CELL_RB201_TESTER_SOCKET_D02                        :=          51132       ,
CELL_RB201_TESTER_SOCKET_D03                        :=          51133       ,
CELL_RB201_TESTER_SOCKET_D04                        :=          51134       ,
CELL_RB201_AP                                       :=          51150       ,
CELL_RB201_AP_TH_A01                                :=          51151       ,
CELL_RB201_AP_TH_A02                                :=          51152       ,
CELL_RB201_AP_TH_A03                                :=          51153       ,
CELL_RB201_AP_TH_A04                                :=          51154       ,
CELL_RB201_AP_TH_B01                                :=          51161       ,
CELL_RB201_AP_TH_B02                                :=          51162       ,
CELL_RB201_AP_TH_B03                                :=          51163       ,
CELL_RB201_AP_TH_B04                                :=          51164       ,
CELL_RB201_AP_TH_C01                                :=          51171       ,
CELL_RB201_AP_TH_C02                                :=          51172       ,
CELL_RB201_AP_TH_C03                                :=          51173       ,
CELL_RB201_AP_TH_C04                                :=          51174       ,
CELL_RB201_AP_TH_D01                                :=          51181       ,
CELL_RB201_AP_TH_D02                                :=          51182       ,
CELL_RB201_AP_TH_D03                                :=          51183       ,
CELL_RB201_AP_TH_D04                                :=          51184       ,
CELL_RB301_TESTER                                   :=          51200       ,
CELL_RB301_TESTER_SOCKET_A01                        :=          51201       ,
CELL_RB301_TESTER_SOCKET_A02                        :=          51202       ,
CELL_RB301_TESTER_SOCKET_A03                        :=          51203       ,
CELL_RB301_TESTER_SOCKET_A04                        :=          51204       ,
CELL_RB301_TESTER_SOCKET_B01                        :=          51211       ,
CELL_RB301_TESTER_SOCKET_B02                        :=          51212       ,
CELL_RB301_TESTER_SOCKET_B03                        :=          51213       ,
CELL_RB301_TESTER_SOCKET_B04                        :=          51214       ,
CELL_RB301_TESTER_SOCKET_C01                        :=          51221       ,
CELL_RB301_TESTER_SOCKET_C02                        :=          51222       ,
CELL_RB301_TESTER_SOCKET_C03                        :=          51223       ,
CELL_RB301_TESTER_SOCKET_C04                        :=          51224       ,
CELL_RB301_TESTER_SOCKET_D01                        :=          51231       ,
CELL_RB301_TESTER_SOCKET_D02                        :=          51232       ,
CELL_RB301_TESTER_SOCKET_D03                        :=          51233       ,
CELL_RB301_TESTER_SOCKET_D04                        :=          51234       ,
CELL_RB301_AP                                       :=          51250       ,
CELL_RB301_AP_TH_A01                                :=          51251       ,
CELL_RB301_AP_TH_A02                                :=          51252       ,
CELL_RB301_AP_TH_A03                                :=          51253       ,
CELL_RB301_AP_TH_A04                                :=          51254       ,
CELL_RB301_AP_TH_B01                                :=          51261       ,
CELL_RB301_AP_TH_B02                                :=          51262       ,
CELL_RB301_AP_TH_B03                                :=          51263       ,
CELL_RB301_AP_TH_B04                                :=          51264       ,
CELL_RB301_AP_TH_C01                                :=          51271       ,
CELL_RB301_AP_TH_C02                                :=          51272       ,
CELL_RB301_AP_TH_C03                                :=          51273       ,
CELL_RB301_AP_TH_C04                                :=          51274       ,
CELL_RB301_AP_TH_D01                                :=          51281       ,
CELL_RB301_AP_TH_D02                                :=          51282       ,
CELL_RB301_AP_TH_D03                                :=          51283       ,
CELL_RB301_AP_TH_D04                                :=          51284       ,
CELL_RB401_TESTER                                   :=          51300       ,
CELL_RB401_TESTER_SOCKET_A01                        :=          51301       ,
CELL_RB401_TESTER_SOCKET_A02                        :=          51302       ,
CELL_RB401_TESTER_SOCKET_A03                        :=          51303       ,
CELL_RB401_TESTER_SOCKET_A04                        :=          51304       ,
CELL_RB401_TESTER_SOCKET_B01                        :=          51311       ,
CELL_RB401_TESTER_SOCKET_B02                        :=          51312       ,
CELL_RB401_TESTER_SOCKET_B03                        :=          51313       ,
CELL_RB401_TESTER_SOCKET_B04                        :=          51314       ,
CELL_RB401_TESTER_SOCKET_C01                        :=          51321       ,
CELL_RB401_TESTER_SOCKET_C02                        :=          51322       ,
CELL_RB401_TESTER_SOCKET_C03                        :=          51323       ,
CELL_RB401_TESTER_SOCKET_C04                        :=          51324       ,
CELL_RB401_TESTER_SOCKET_D01                        :=          51331       ,
CELL_RB401_TESTER_SOCKET_D02                        :=          51332       ,
CELL_RB401_TESTER_SOCKET_D03                        :=          51333       ,
CELL_RB401_TESTER_SOCKET_D04                        :=          51334       ,
CELL_RB401_AP                                       :=          51350       ,
CELL_RB401_AP_TH_A01                                :=          51351       ,
CELL_RB401_AP_TH_A02                                :=          51352       ,
CELL_RB401_AP_TH_A03                                :=          51353       ,
CELL_RB401_AP_TH_A04                                :=          51354       ,
CELL_RB401_AP_TH_B01                                :=          51361       ,
CELL_RB401_AP_TH_B02                                :=          51362       ,
CELL_RB401_AP_TH_B03                                :=          51363       ,
CELL_RB401_AP_TH_B04                                :=          51364       ,
CELL_RB401_AP_TH_C01                                :=          51371       ,
CELL_RB401_AP_TH_C02                                :=          51372       ,
CELL_RB401_AP_TH_C03                                :=          51373       ,
CELL_RB401_AP_TH_C04                                :=          51374       ,
CELL_RB401_AP_TH_D01                                :=          51381       ,
CELL_RB401_AP_TH_D02                                :=          51382       ,
CELL_RB401_AP_TH_D03                                :=          51383       ,
CELL_RB401_AP_TH_D04                                :=          51384       ,
CELL_RB501_TESTER                                   :=          51400       ,
CELL_RB501_TESTER_SOCKET_A01                        :=          51401       ,
CELL_RB501_TESTER_SOCKET_A02                        :=          51402       ,
CELL_RB501_TESTER_SOCKET_A03                        :=          51403       ,
CELL_RB501_TESTER_SOCKET_A04                        :=          51404       ,
CELL_RB501_TESTER_SOCKET_B01                        :=          51411       ,
CELL_RB501_TESTER_SOCKET_B02                        :=          51412       ,
CELL_RB501_TESTER_SOCKET_B03                        :=          51413       ,
CELL_RB501_TESTER_SOCKET_B04                        :=          51414       ,
CELL_RB501_TESTER_SOCKET_C01                        :=          51421       ,
CELL_RB501_TESTER_SOCKET_C02                        :=          51422       ,
CELL_RB501_TESTER_SOCKET_C03                        :=          51423       ,
CELL_RB501_TESTER_SOCKET_C04                        :=          51424       ,
CELL_RB501_TESTER_SOCKET_D01                        :=          51431       ,
CELL_RB501_TESTER_SOCKET_D02                        :=          51432       ,
CELL_RB501_TESTER_SOCKET_D03                        :=          51433       ,
CELL_RB501_TESTER_SOCKET_D04                        :=          51434       ,
CELL_RB501_AP                                       :=          51450       ,
CELL_RB501_AP_TH_A01                                :=          51451       ,
CELL_RB501_AP_TH_A02                                :=          51452       ,
CELL_RB501_AP_TH_A03                                :=          51453       ,
CELL_RB501_AP_TH_A04                                :=          51454       ,
CELL_RB501_AP_TH_B01                                :=          51461       ,
CELL_RB501_AP_TH_B02                                :=          51462       ,
CELL_RB501_AP_TH_B03                                :=          51463       ,
CELL_RB501_AP_TH_B04                                :=          51464       ,
CELL_RB501_AP_TH_C01                                :=          51471       ,
CELL_RB501_AP_TH_C02                                :=          51472       ,
CELL_RB501_AP_TH_C03                                :=          51473       ,
CELL_RB501_AP_TH_C04                                :=          51474       ,
CELL_RB501_AP_TH_D01                                :=          51481       ,
CELL_RB501_AP_TH_D02                                :=          51482       ,
CELL_RB501_AP_TH_D03                                :=          51483       ,
CELL_RB501_AP_TH_D04                                :=          51484       ,
CELL_RB601_TESTER                                   :=          51500       ,
CELL_RB601_TESTER_SOCKET_A01                        :=          51501       ,
CELL_RB601_TESTER_SOCKET_A02                        :=          51502       ,
CELL_RB601_TESTER_SOCKET_A03                        :=          51503       ,
CELL_RB601_TESTER_SOCKET_A04                        :=          51504       ,
CELL_RB601_TESTER_SOCKET_B01                        :=          51511       ,
CELL_RB601_TESTER_SOCKET_B02                        :=          51512       ,
CELL_RB601_TESTER_SOCKET_B03                        :=          51513       ,
CELL_RB601_TESTER_SOCKET_B04                        :=          51514       ,
CELL_RB601_TESTER_SOCKET_C01                        :=          51521       ,
CELL_RB601_TESTER_SOCKET_C02                        :=          51522       ,
CELL_RB601_TESTER_SOCKET_C03                        :=          51523       ,
CELL_RB601_TESTER_SOCKET_C04                        :=          51524       ,
CELL_RB601_TESTER_SOCKET_D01                        :=          51531       ,
CELL_RB601_TESTER_SOCKET_D02                        :=          51532       ,
CELL_RB601_TESTER_SOCKET_D03                        :=          51533       ,
CELL_RB601_TESTER_SOCKET_D04                        :=          51534       ,
CELL_RB601_AP                                       :=          51550       ,
CELL_RB601_AP_TH_A01                                :=          51551       ,
CELL_RB601_AP_TH_A02                                :=          51552       ,
CELL_RB601_AP_TH_A03                                :=          51553       ,
CELL_RB601_AP_TH_A04                                :=          51554       ,
CELL_RB601_AP_TH_B01                                :=          51561       ,
CELL_RB601_AP_TH_B02                                :=          51562       ,
CELL_RB601_AP_TH_B03                                :=          51563       ,
CELL_RB601_AP_TH_B04                                :=          51564       ,
CELL_RB601_AP_TH_C01                                :=          51571       ,
CELL_RB601_AP_TH_C02                                :=          51572       ,
CELL_RB601_AP_TH_C03                                :=          51573       ,
CELL_RB601_AP_TH_C04                                :=          51574       ,
CELL_RB601_AP_TH_D01                                :=          51581       ,
CELL_RB601_AP_TH_D02                                :=          51582       ,
CELL_RB601_AP_TH_D03                                :=          51583       ,
CELL_RB601_AP_TH_D04                                :=          51584       ,
CELL_RC101_TESTER                                   :=          52000       ,
CELL_RC101_TESTER_SOCKET_A01                        :=          52001       ,
CELL_RC101_TESTER_SOCKET_A02                        :=          52002       ,
CELL_RC101_TESTER_SOCKET_A03                        :=          52003       ,
CELL_RC101_TESTER_SOCKET_A04                        :=          52004       ,
CELL_RC101_TESTER_SOCKET_B01                        :=          52011       ,
CELL_RC101_TESTER_SOCKET_B02                        :=          52012       ,
CELL_RC101_TESTER_SOCKET_B03                        :=          52013       ,
CELL_RC101_TESTER_SOCKET_B04                        :=          52014       ,
CELL_RC101_TESTER_SOCKET_C01                        :=          52021       ,
CELL_RC101_TESTER_SOCKET_C02                        :=          52022       ,
CELL_RC101_TESTER_SOCKET_C03                        :=          52023       ,
CELL_RC101_TESTER_SOCKET_C04                        :=          52024       ,
CELL_RC101_TESTER_SOCKET_D01                        :=          52031       ,
CELL_RC101_TESTER_SOCKET_D02                        :=          52032       ,
CELL_RC101_TESTER_SOCKET_D03                        :=          52033       ,
CELL_RC101_TESTER_SOCKET_D04                        :=          52034       ,
CELL_RC101_AP                                       :=          52050       ,
CELL_RC101_AP_TH_A01                                :=          52051       ,
CELL_RC101_AP_TH_A02                                :=          52052       ,
CELL_RC101_AP_TH_A03                                :=          52053       ,
CELL_RC101_AP_TH_A04                                :=          52054       ,
CELL_RC101_AP_TH_B01                                :=          52061       ,
CELL_RC101_AP_TH_B02                                :=          52062       ,
CELL_RC101_AP_TH_B03                                :=          52063       ,
CELL_RC101_AP_TH_B04                                :=          52064       ,
CELL_RC101_AP_TH_C01                                :=          52071       ,
CELL_RC101_AP_TH_C02                                :=          52072       ,
CELL_RC101_AP_TH_C03                                :=          52073       ,
CELL_RC101_AP_TH_C04                                :=          52074       ,
CELL_RC101_AP_TH_D01                                :=          52081       ,
CELL_RC101_AP_TH_D02                                :=          52082       ,
CELL_RC101_AP_TH_D03                                :=          52083       ,
CELL_RC101_AP_TH_D04                                :=          52084       ,
CELL_RC201_TESTER                                   :=          52100       ,
CELL_RC201_TESTER_SOCKET_A01                        :=          52101       ,
CELL_RC201_TESTER_SOCKET_A02                        :=          52102       ,
CELL_RC201_TESTER_SOCKET_A03                        :=          52103       ,
CELL_RC201_TESTER_SOCKET_A04                        :=          52104       ,
CELL_RC201_TESTER_SOCKET_B01                        :=          52111       ,
CELL_RC201_TESTER_SOCKET_B02                        :=          52112       ,
CELL_RC201_TESTER_SOCKET_B03                        :=          52113       ,
CELL_RC201_TESTER_SOCKET_B04                        :=          52114       ,
CELL_RC201_TESTER_SOCKET_C01                        :=          52121       ,
CELL_RC201_TESTER_SOCKET_C02                        :=          52122       ,
CELL_RC201_TESTER_SOCKET_C03                        :=          52123       ,
CELL_RC201_TESTER_SOCKET_C04                        :=          52124       ,
CELL_RC201_TESTER_SOCKET_D01                        :=          52131       ,
CELL_RC201_TESTER_SOCKET_D02                        :=          52132       ,
CELL_RC201_TESTER_SOCKET_D03                        :=          52133       ,
CELL_RC201_TESTER_SOCKET_D04                        :=          52134       ,
CELL_RC201_AP                                       :=          52150       ,
CELL_RC201_AP_TH_A01                                :=          52151       ,
CELL_RC201_AP_TH_A02                                :=          52152       ,
CELL_RC201_AP_TH_A03                                :=          52153       ,
CELL_RC201_AP_TH_A04                                :=          52154       ,
CELL_RC201_AP_TH_B01                                :=          52161       ,
CELL_RC201_AP_TH_B02                                :=          52162       ,
CELL_RC201_AP_TH_B03                                :=          52163       ,
CELL_RC201_AP_TH_B04                                :=          52164       ,
CELL_RC201_AP_TH_C01                                :=          52171       ,
CELL_RC201_AP_TH_C02                                :=          52172       ,
CELL_RC201_AP_TH_C03                                :=          52173       ,
CELL_RC201_AP_TH_C04                                :=          52174       ,
CELL_RC201_AP_TH_D01                                :=          52181       ,
CELL_RC201_AP_TH_D02                                :=          52182       ,
CELL_RC201_AP_TH_D03                                :=          52183       ,
CELL_RC201_AP_TH_D04                                :=          52184       ,
CELL_RC301_TESTER                                   :=          52200       ,
CELL_RC301_TESTER_SOCKET_A01                        :=          52201       ,
CELL_RC301_TESTER_SOCKET_A02                        :=          52202       ,
CELL_RC301_TESTER_SOCKET_A03                        :=          52203       ,
CELL_RC301_TESTER_SOCKET_A04                        :=          52204       ,
CELL_RC301_TESTER_SOCKET_B01                        :=          52211       ,
CELL_RC301_TESTER_SOCKET_B02                        :=          52212       ,
CELL_RC301_TESTER_SOCKET_B03                        :=          52213       ,
CELL_RC301_TESTER_SOCKET_B04                        :=          52214       ,
CELL_RC301_TESTER_SOCKET_C01                        :=          52221       ,
CELL_RC301_TESTER_SOCKET_C02                        :=          52222       ,
CELL_RC301_TESTER_SOCKET_C03                        :=          52223       ,
CELL_RC301_TESTER_SOCKET_C04                        :=          52224       ,
CELL_RC301_TESTER_SOCKET_D01                        :=          52231       ,
CELL_RC301_TESTER_SOCKET_D02                        :=          52232       ,
CELL_RC301_TESTER_SOCKET_D03                        :=          52233       ,
CELL_RC301_TESTER_SOCKET_D04                        :=          52234       ,
CELL_RC301_AP                                       :=          52250       ,
CELL_RC301_AP_TH_A01                                :=          52251       ,
CELL_RC301_AP_TH_A02                                :=          52252       ,
CELL_RC301_AP_TH_A03                                :=          52253       ,
CELL_RC301_AP_TH_A04                                :=          52254       ,
CELL_RC301_AP_TH_B01                                :=          52261       ,
CELL_RC301_AP_TH_B02                                :=          52262       ,
CELL_RC301_AP_TH_B03                                :=          52263       ,
CELL_RC301_AP_TH_B04                                :=          52264       ,
CELL_RC301_AP_TH_C01                                :=          52271       ,
CELL_RC301_AP_TH_C02                                :=          52272       ,
CELL_RC301_AP_TH_C03                                :=          52273       ,
CELL_RC301_AP_TH_C04                                :=          52274       ,
CELL_RC301_AP_TH_D01                                :=          52281       ,
CELL_RC301_AP_TH_D02                                :=          52282       ,
CELL_RC301_AP_TH_D03                                :=          52283       ,
CELL_RC301_AP_TH_D04                                :=          52284       ,
CELL_RC401_TESTER                                   :=          52300       ,
CELL_RC401_TESTER_SOCKET_A01                        :=          52301       ,
CELL_RC401_TESTER_SOCKET_A02                        :=          52302       ,
CELL_RC401_TESTER_SOCKET_A03				        :=          52303       ,
CELL_RC401_TESTER_SOCKET_A04                        :=          52304       ,
CELL_RC401_TESTER_SOCKET_B01                        :=          52311       ,
CELL_RC401_TESTER_SOCKET_B02                        :=          52312       ,
CELL_RC401_TESTER_SOCKET_B03                        :=          52313       ,
CELL_RC401_TESTER_SOCKET_B04                        :=          52314       ,
CELL_RC401_TESTER_SOCKET_C01                        :=          52321       ,
CELL_RC401_TESTER_SOCKET_C02                        :=          52322       ,
CELL_RC401_TESTER_SOCKET_C03                        :=          52323       ,
CELL_RC401_TESTER_SOCKET_C04                        :=          52324       ,
CELL_RC401_TESTER_SOCKET_D01                        :=          52331       ,
CELL_RC401_TESTER_SOCKET_D02                        :=          52332       ,
CELL_RC401_TESTER_SOCKET_D03                        :=          52333       ,
CELL_RC401_TESTER_SOCKET_D04                        :=          52334       ,
CELL_RC401_AP                                       :=          52350       ,
CELL_RC401_AP_TH_A01                                :=          52351       ,
CELL_RC401_AP_TH_A02                                :=          52352       ,
CELL_RC401_AP_TH_A03                                :=          52353       ,
CELL_RC401_AP_TH_A04                                :=          52354       ,
CELL_RC401_AP_TH_B01                                :=          52361       ,
CELL_RC401_AP_TH_B02                                :=          52362       ,
CELL_RC401_AP_TH_B03                                :=          52363       ,
CELL_RC401_AP_TH_B04                                :=          52364       ,
CELL_RC401_AP_TH_C01                                :=          52371       ,
CELL_RC401_AP_TH_C02                                :=          52372       ,
CELL_RC401_AP_TH_C03                                :=          52373       ,
CELL_RC401_AP_TH_C04                                :=          52374       ,
CELL_RC401_AP_TH_D01                                :=          52381       ,
CELL_RC401_AP_TH_D02                                :=          52382       ,
CELL_RC401_AP_TH_D03                                :=          52383       ,
CELL_RC401_AP_TH_D04                                :=          52384       ,
CELL_RC501_TESTER                                   :=          52400       ,
CELL_RC501_TESTER_SOCKET_A01                        :=          52401       ,
CELL_RC501_TESTER_SOCKET_A02                        :=          52402       ,
CELL_RC501_TESTER_SOCKET_A03                        :=          52403       ,
CELL_RC501_TESTER_SOCKET_A04                        :=          52404       ,
CELL_RC501_TESTER_SOCKET_B01                        :=          52411       ,
CELL_RC501_TESTER_SOCKET_B02                        :=          52412       ,
CELL_RC501_TESTER_SOCKET_B03                        :=          52413       ,
CELL_RC501_TESTER_SOCKET_B04                        :=          52414       ,
CELL_RC501_TESTER_SOCKET_C01                        :=          52421       ,
CELL_RC501_TESTER_SOCKET_C02                        :=          52422       ,
CELL_RC501_TESTER_SOCKET_C03                        :=          52423       ,
CELL_RC501_TESTER_SOCKET_C04                        :=          52424       ,
CELL_RC501_TESTER_SOCKET_D01                        :=          52431       ,
CELL_RC501_TESTER_SOCKET_D02                        :=          52432       ,
CELL_RC501_TESTER_SOCKET_D03                        :=          52433       ,
CELL_RC501_TESTER_SOCKET_D04                        :=          52434       ,
CELL_RC501_AP                                       :=          52450       ,
CELL_RC501_AP_TH_A01                                :=          52451       ,
CELL_RC501_AP_TH_A02                                :=          52452       ,
CELL_RC501_AP_TH_A03                                :=          52453       ,
CELL_RC501_AP_TH_A04                                :=          52454       ,
CELL_RC501_AP_TH_B01                                :=          52461       ,
CELL_RC501_AP_TH_B02                                :=          52462       ,
CELL_RC501_AP_TH_B03                                :=          52463       ,
CELL_RC501_AP_TH_B04                                :=          52464       ,
CELL_RC501_AP_TH_C01                                :=          52471       ,
CELL_RC501_AP_TH_C02                                :=          52472       ,
CELL_RC501_AP_TH_C03                                :=          52473       ,
CELL_RC501_AP_TH_C04                                :=          52474       ,
CELL_RC501_AP_TH_D01                                :=          52481       ,
CELL_RC501_AP_TH_D02                                :=          52482       ,
CELL_RC501_AP_TH_D03                                :=          52483       ,
CELL_RC501_AP_TH_D04                                :=          52484       ,
CELL_RC601_TESTER                                   :=          52500       ,
CELL_RC601_TESTER_SOCKET_A01                        :=          52501       ,
CELL_RC601_TESTER_SOCKET_A02                        :=          52502       ,
CELL_RC601_TESTER_SOCKET_A03                        :=          52503       ,
CELL_RC601_TESTER_SOCKET_A04                        :=          52504       ,
CELL_RC601_TESTER_SOCKET_B01                        :=          52511       ,
CELL_RC601_TESTER_SOCKET_B02                        :=          52512       ,
CELL_RC601_TESTER_SOCKET_B03                        :=          52513       ,
CELL_RC601_TESTER_SOCKET_B04                        :=          52514       ,
CELL_RC601_TESTER_SOCKET_C01                        :=          52521       ,
CELL_RC601_TESTER_SOCKET_C02                        :=          52522       ,
CELL_RC601_TESTER_SOCKET_C03                        :=          52523       ,
CELL_RC601_TESTER_SOCKET_C04                        :=          52524       ,
CELL_RC601_TESTER_SOCKET_D01                        :=          52531       ,
CELL_RC601_TESTER_SOCKET_D02                        :=          52532       ,
CELL_RC601_TESTER_SOCKET_D03                        :=          52533       ,
CELL_RC601_TESTER_SOCKET_D04                        :=          52534       ,
CELL_RC601_AP                                       :=          52550       ,
CELL_RC601_AP_TH_A01                                :=          52551       ,
CELL_RC601_AP_TH_A02                                :=          52552       ,
CELL_RC601_AP_TH_A03                                :=          52553       ,
CELL_RC601_AP_TH_A04                                :=          52554       ,
CELL_RC601_AP_TH_B01                                :=          52561       ,
CELL_RC601_AP_TH_B02                                :=          52562       ,
CELL_RC601_AP_TH_B03                                :=          52563       ,
CELL_RC601_AP_TH_B04                                :=          52564       ,
CELL_RC601_AP_TH_C01                                :=          52571       ,
CELL_RC601_AP_TH_C02                                :=          52572       ,
CELL_RC601_AP_TH_C03                                :=          52573       ,
CELL_RC601_AP_TH_C04                                :=          52574       ,
CELL_RC601_AP_TH_D01                                :=          52581       ,
CELL_RC601_AP_TH_D02                                :=          52582       ,
CELL_RC601_AP_TH_D03                                :=          52583       ,
CELL_RC601_AP_TH_D04                                :=          52584       ,
CELL_LA101_TIERII                                   :=          54090       ,
CELL_LA201_TIERII                                   :=          54091       ,
CELL_LA301_TIERII                                   :=          54092       ,
CELL_LA401_TIERII                                   :=          54093       ,
CELL_LA501_TIERII                                   :=          54094       ,
CELL_LA601_TIERII                                   :=          54095       ,
CELL_LB101_TIERII                                   :=          54096       ,
CELL_LB201_TIERII                                   :=          54097       ,
CELL_LB301_TIERII                                   :=          54098       ,
CELL_LB401_TIERII                                   :=          54099       ,
CELL_LB501_TIERII                                   :=          54100       ,
CELL_LB601_TIERII                                   :=          54101       ,
CELL_LC101_TIERII                                   :=          54102       ,
CELL_LC201_TIERII                                   :=          54103       ,
CELL_LC301_TIERII                                   :=          54104       ,
CELL_LC401_TIERII                                   :=          54105       ,
CELL_LC501_TIERII                                   :=          54106       ,
CELL_LC601_TIERII                                   :=          54107       ,
CELL_RA101_TIERII                                   :=          54108       ,
CELL_RA201_TIERII                                   :=          54109       ,
CELL_RA301_TIERII                                   :=          54110       ,
CELL_RA401_TIERII                                   :=          54111       ,
CELL_RA501_TIERII                                   :=          54112       ,
CELL_RA601_TIERII                                   :=          54113       ,
CELL_RB101_TIERII                                   :=          54114       ,
CELL_RB201_TIERII                                   :=          54115       ,
CELL_RB301_TIERII                                   :=          54116       ,
CELL_RB401_TIERII                                   :=          54117       ,
CELL_RB501_TIERII                                   :=          54118       ,
CELL_RB601_TIERII                                   :=          54119       ,
CELL_RC101_TIERII                                   :=          54120       ,
CELL_RC201_TIERII                                   :=          54121       ,
CELL_RC301_TIERII                                   :=          54122       ,
CELL_RC401_TIERII                                   :=          54123       ,
CELL_RC501_TIERII                                   :=          54124       ,
CELL_RC601_TIERII                                   :=          54125       

(*
	//New 												  
	NA                                              :=      0    		,
	Standby                                         :=      1           ,
	IOLP                                            :=      2           ,
	PNB                                             :=      3           ,
	TBOT                                            :=      4           ,
	LP_VISIONSHUTTLE_L                              :=      1500        ,
	LP_VISIONSHUTTLE_R                              :=      1600        ,
	LP_LE                                           :=      1900        ,
	LP_L01                                          :=      1901        ,
	LP_L02                                          :=      1902        ,
	LP_RE                                           :=      1903        ,
	LP_R01                                          :=      1904        ,
	LP_R02                                          :=      1905        ,
	LP_L                                            :=      1910        ,
	LP_R                                            :=      1911        ,
	LP_LE_STACKER_01                                :=      2000        ,
	LP_LE_STACKER_01_LIFT                           :=      2001        ,
	LP_LE_STACKER_01_STOPPER_01                     :=      2002        ,
	LP_LE_STACKER_01_STOPPER_02                     :=      2003        ,
	LP_LE_STACKER_02                                :=      2050        ,
	LP_LE_STACKER_02_LIFT                           :=      2051        ,
	LP_LE_STACKER_02_STOPPER_01                     :=      2052        ,
	LP_LE_STACKER_02_STOPPER_02                     :=      2053        ,
	LP_LE_CONVEYOR                                  :=      2200        ,
	LP_LE_CONVEYOR_STACKER_01_PRE                   :=      2250        ,
	LP_LE_CONVEYOR_STACKER_01                       :=      2251        ,
	LP_LE_CONVEYOR_STACKER_01_POST                  :=      2252        ,
	LP_LE_CONVEYOR_STACKER_02                       :=      2300        ,
	LP_L01_STACKER_01                               :=      3000        ,
	LP_L01_STACKER_01_LIFT                          :=      3001        ,
	LP_L01_STACKER_01_STOPPER_01                    :=      3002        ,
	LP_L01_STACKER_01_STOPPER_02                    :=      3003        ,
	LP_L01_STACKER_02                               :=      3050        ,
	LP_L01_STACKER_02_LIFT                          :=      3051        ,
	LP_L01_STACKER_02_STOPPER_01                    :=      3052        ,
	LP_L01_STACKER_02_STOPPER_02                    :=      3053        ,
	LP_L01_STACKER_03                               :=      3100        ,
	LP_L01_STACKER_03_LIFT                          :=      3101        ,
	LP_L01_STACKER_03_STOPPER_01                    :=      3102        ,
	LP_L01_STACKER_03_STOPPER_02                    :=      3103        ,
	LP_L01_CONVEYOR_01                              :=      3110        ,
	LP_L01_CONVEYOR_02                              :=      3120        ,
	LP_L01_CONVEYOR_STACKER_01_PRE                  :=      3125        ,
	LP_L01_CONVEYOR_STACKER_01                      :=      3126        ,
	LP_L01_CONVEYOR_STACKER_01_POST                 :=      3127        ,
	LP_L01_CONVEYOR_STACKER_02                      :=      3128        ,
	LP_L01_CONVEYOR_STACKER_02_POST                 :=      3129        ,
	LP_L01_EPORT                                    :=      3130        ,
	LP_L01_EPORT_STANDBY                            :=      3131        ,
	LP_L01_EPORT_STOPPER_01                         :=      3132        ,
	LP_L01_EPORT_STOPPER_02                         :=      3133        ,
	LP_L01_VISION                                   :=      3140        ,
	LP_L01_UPORT                                    :=      3151        ,
	LP_L02_STACKER_01                               :=      3200        ,
	LP_L02_STACKER_01_LIFT                          :=      3201        ,
	LP_L02_STACKER_01_STOPPER_01                    :=      3202        ,
	LP_L02_STACKER_01_STOPPER_02                    :=      3203        ,
	LP_L02_STACKER_02                               :=      3250        ,
	LP_L02_STACKER_02_LIFT                          :=      3251        ,
	LP_L02_STACKER_02_STOPPER_01                    :=      3252        ,
	LP_L02_STACKER_02_STOPPER_02                    :=      3253        ,
	LP_L02_STACKER_03                               :=      3300        ,
	LP_L02_STACKER_03_LIFT                          :=      3301        ,
	LP_L02_STACKER_03_STOPPER_01                    :=      3302        ,
	LP_L02_STACKER_03_STOPPER_02                    :=      3303        ,
	LP_L02_CONVEYOR_01                              :=      3310        ,
	LP_L02_CONVEYOR_02                              :=      3320        ,
	LP_L02_CONVEYOR_STACKER_01_PRE                  :=      3325        ,
	LP_L02_CONVEYOR_STACKER_01                      :=      3326        ,
	LP_L02_CONVEYOR_STACKER_01_POST                 :=      3327        ,
	LP_L02_CONVEYOR_STACKER_02                      :=      3328        ,
	LP_L02_CONVEYOR_STACKER_02_POST                 :=      3329        ,
	LP_L02_EPORT                                    :=      3330        ,
	LP_L02_EPORT_STANDBY                            :=      3331        ,
	LP_L02_EPORT_STOPPER_01                         :=      3332        ,
	LP_L02_EPORT_STOPPER_02                         :=      3333        ,
	LP_L02_VISION                                   :=      3340        ,
	LP_L02_UPORT                                    :=      3351        ,
	LP_RE_STACKER_01                                :=      4000        ,
	LP_RE_STACKER_01_LIFT                           :=      4001        ,
	LP_RE_STACKER_01_STOPPER_01                     :=      4002        ,
	LP_RE_STACKER_01_STOPPER_02                     :=      4003        ,
	LP_RE_STACKER_02                                :=      4050        ,
	LP_RE_STACKER_02_LIFT                           :=      4051        ,
	LP_RE_STACKER_02_STOPPER_01                     :=      4052        ,
	LP_RE_STACKER_02_STOPPER_02                     :=      4053        ,
	LP_RE_CONVEYOR                                  :=      4200        ,
	LP_RE_CONVEYOR_STACKER_01_PRE                   :=      4250        ,
	LP_RE_CONVEYOR_STACKER_01                       :=      4251        ,
	LP_RE_CONVEYOR_STACKER_01_POST                  :=      4252        ,
	LP_RE_CONVEYOR_STACKER_02                       :=      4300        ,
	LP_R01_STACKER_01                               :=      5000        ,
	LP_R01_STACKER_01_LIFT                          :=      5001        ,
	LP_R01_STACKER_01_STOPPER_01                    :=      5002        ,
	LP_R01_STACKER_01_STOPPER_02                    :=      5003        ,
	LP_R01_STACKER_02                               :=      5050        ,
	LP_R01_STACKER_02_LIFT                          :=      5051        ,
	LP_R01_STACKER_02_STOPPER_01                    :=      5052        ,
	LP_R01_STACKER_02_STOPPER_02                    :=      5053        ,
	LP_R01_STACKER_03                               :=      5100        ,
	LP_R01_STACKER_03_LIFT                          :=      5101        ,
	LP_R01_STACKER_03_STOPPER_01                    :=      5102        ,
	LP_R01_STACKER_03_STOPPER_02                    :=      5103        ,
	LP_R01_CONVEYOR_01                              :=      5110        ,
	LP_R01_CONVEYOR_02                              :=      5120        ,
	LP_R01_CONVEYOR_STACKER_01_PRE                  :=      5125        ,
	LP_R01_CONVEYOR_STACKER_01                      :=      5126        ,
	LP_R01_CONVEYOR_STACKER_01_POST                 :=      5127        ,
	LP_R01_CONVEYOR_STACKER_02                      :=      5128        ,
	LP_R01_CONVEYOR_STACKER_02_POST                 :=      5129        ,
	LP_R01_EPORT                                    :=      5130        ,
	LP_R01_EPORT_STANDBY                            :=      5131        ,
	LP_R01_EPORT_STOPPER_01                         :=      5132        ,
	LP_R01_EPORT_STOPPER_02                         :=      5133        ,
	LP_R01_VISION                                   :=      5140        ,
	LP_R01_UPORT                                    :=      5151        ,
	LP_R02_STACKER_01                               :=      5200        ,
	LP_R02_STACKER_01_LIFT                          :=      5201        ,
	LP_R02_STACKER_01_STOPPER_01                    :=      5202        ,
	LP_R02_STACKER_01_STOPPER_02                    :=      5203        ,
	LP_R02_STACKER_02                               :=      5250        ,
	LP_R02_STACKER_02_LIFT                          :=      5251        ,
	LP_R02_STACKER_02_STOPPER_01                    :=      5252        ,
	LP_R02_STACKER_02_STOPPER_02                    :=      5253        ,
	LP_R02_STACKER_03                               :=      5300        ,
	LP_R02_STACKER_03_LIFT                          :=      5301        ,
	LP_R02_STACKER_03_STOPPER_01                    :=      5302        ,
	LP_R02_STACKER_03_STOPPER_02                    :=      5303        ,
	LP_R02_CONVEYOR_01                              :=      5310        ,
	LP_R02_CONVEYOR_02                              :=      5320        ,
	LP_R02_CONVEYOR_STACKER_01_PRE                  :=      5325        ,
	LP_R02_CONVEYOR_STACKER_01                      :=      5326        ,
	LP_R02_CONVEYOR_STACKER_01_POST                 :=      5327        ,
	LP_R02_CONVEYOR_STACKER_02                      :=      5328        ,
	LP_R02_CONVEYOR_STACKER_02_POST                 :=      5329        ,
	LP_R02_EPORT                                    :=      5330        ,
	LP_R02_EPORT_STANDBY                            :=      5331        ,
	LP_R02_EPORT_STOPPER_01                         :=      5332        ,
	LP_R02_EPORT_STOPPER_02                         :=      5333        ,
	LP_R02_VISION                                   :=      5340        ,
	LP_R02_UPORT                                    :=      5351        ,
	TTS                                             :=      10000       ,
	TTS_SHUTTLE_01                                  :=      10100       ,
	TTS_SHUTTLE_01_SERVICE                          :=      10101       ,
	TTS_SHUTTLE_01_PARK                             :=      10102       ,
	TTS_SHUTTLE_01_CONVEYOR                         :=      10103       ,
	TTS_SHUTTLE_02                                  :=      10200       ,
	TTS_SHUTTLE_02_SERVICE                          :=      10201       ,
	TTS_SHUTTLE_02_CONVEYOR                         :=      10202       ,
	TTS_SHUTTLE_03                                  :=      10300       ,
	TTS_SHUTTLE_03_SERVICE                          :=      10301       ,
	TTS_SHUTTLE_03_PARK                             :=      10302       ,
	TTS_SHUTTLE_03_CONVEYOR                         :=      10303       ,
	PNB_DOOR_TOP_LEFT                               :=      20001       ,
	PNB_DOOR_TOP_RIGHT                              :=      20002       ,
	PNB_DOOR_BOTTOM                                 :=      20003       ,
	PNB_LANE_01                                     :=      21000       ,
	PNB_LANE_01_CONVEYOR                            :=      21001       ,
	PNB_LANE_02                                     :=      21050       ,
	PNB_LANE_02_CONVEYOR                            :=      21051       ,
	PNB_LANE_03                                     :=      21150       ,
	PNB_LANE_03_CONVEYOR                            :=      21151       ,
	PNB_LANE_04                                     :=      21200       ,
	PNB_LANE_04_CONVEYOR                            :=      21201       ,
	PNB_LANE_05                                     :=      21350       ,
	PNB_LANE_05_CONVEYOR                            :=      21351       ,
	PNB_LANE_06                                     :=      21400       ,
	PNB_LANE_06_CONVEYOR                            :=      21401       ,
	PNB_LANE_07                                     :=      21450       ,
	PNB_LANE_07_CONVEYOR                            :=      21451       ,
	PNB_LANE_08                                     :=      21500       ,
	PNB_LANE_08_CONVEYOR                            :=      21501       ,
	PNB_GANTRY_01                                   :=      22500       ,
	PNB_GANTRY_01_PARK                              :=      22501       ,
	PNB_UPCAM_L                                     :=      22502       ,
	PNB_RFID_L                                      :=      22503       ,
	PNB_RFID_L_01                                   :=      22504       ,
	PNB_RFID_L_02                                   :=      22505       ,
	PNB_GANTRY_01_SERVICE                           :=      22506       ,
	PNB_GANTRY_01_HEAD_A01                          :=      22550       ,
	PNB_GANTRY_01_HEAD_A02                          :=      22560       ,
	PNB_GANTRY_01_HEAD_A03                          :=      22570       ,
	PNB_GANTRY_01_HEAD_A04                          :=      22580       ,
	PNB_GANTRY_02                                   :=      23000       ,
	PNB_GANTRY_02_PARK                              :=      23001       ,
	PNB_UPCAM_R                                     :=      23002       ,
	PNB_RFID_R                                      :=      23003       ,
	PNB_RFID_R_01                                   :=      23004       ,
	PNB_RFID_R_02                                   :=      23005       ,
	PNB_GANTRY_02_SERVICE                           :=      22506       ,
	PNB_GANTRY_02_HEAD_A01                          :=      23050       ,
	PNB_GANTRY_02_HEAD_A02                          :=      23060       ,
	PNB_GANTRY_02_HEAD_A03                          :=      23070       ,
	PNB_GANTRY_02_HEAD_A04                          :=      23080       ,
	PRECISOR_UL                                     :=      24000       ,
	PRECISOR_UL_CLEAN                               :=      24001       ,
	PRECISOR_UL_01                                  :=      24002       ,
	PRECISOR_UL_02                                  :=      24003       ,
	PRECISOR_UL_CLEAN_READID                        :=      24004       ,
	PRECISOR_UL_01_READID                           :=      24005       ,
	PRECISOR_UL_02_READID                           :=      24006       ,
	PRECISOR_UL_A01_01                              :=      24011       ,
	PRECISOR_UL_A01_02                              :=      24012       ,
	PRECISOR_UL_A02_01                              :=      24021       ,
	PRECISOR_UL_A02_02                              :=      24022       ,
	PRECISOR_UL_A03_01                              :=      24031       ,
	PRECISOR_UL_A03_02                              :=      24032       ,
	PRECISOR_UL_A04_01                              :=      24041       ,
	PRECISOR_UL_A04_02                              :=      24042       ,
	PRECISOR_UL_B01_01                              :=      24061       ,
	PRECISOR_UL_B01_02                              :=      24062       ,
	PRECISOR_UL_B02_01                              :=      24071       ,
	PRECISOR_UL_B02_02                              :=      24072       ,
	PRECISOR_UL_B03_01                              :=      24081       ,
	PRECISOR_UL_B03_02                              :=      24082       ,
	PRECISOR_UL_B04_01                              :=      24091       ,
	PRECISOR_UL_B04_02                              :=      24092       ,
	PRECISOR_UL_C01_01                              :=      24111       ,
	PRECISOR_UL_C01_02                              :=      24112       ,
	PRECISOR_UL_C02_01                              :=      24121       ,
	PRECISOR_UL_C02_02                              :=      24122       ,
	PRECISOR_UL_C03_01                              :=      24131       ,
	PRECISOR_UL_C03_02                              :=      24132       ,
	PRECISOR_UL_C04_01                              :=      24141       ,
	PRECISOR_UL_C04_02                              :=      24142       ,
	PRECISOR_UL_D01_01                              :=      24161       ,
	PRECISOR_UL_D01_02                              :=      24162       ,
	PRECISOR_UL_D02_01                              :=      24171       ,
	PRECISOR_UL_D02_02                              :=      24172       ,
	PRECISOR_UL_D03_01                              :=      24181       ,
	PRECISOR_UL_D03_02                              :=      24182       ,
	PRECISOR_UL_D04_01                              :=      24191       ,
	PRECISOR_UL_D04_02                              :=      24192       ,
	PRECISOR_UR                                     :=      24500       ,
	PRECISOR_UR_CLEAN                               :=      24501       ,
	PRECISOR_UR_01                                  :=      24502       ,
	PRECISOR_UR_02                                  :=      24503       ,
	PRECISOR_UR_CLEAN_READID                        :=      24504       ,
	PRECISOR_UR_01_READID                           :=      24505       ,
	PRECISOR_UR_02_READID                           :=      24506       ,
	PRECISOR_UR_A01_01                              :=      24511       ,
	PRECISOR_UR_A01_02                              :=      24512       ,
	PRECISOR_UR_A02_01                              :=      24521       ,
	PRECISOR_UR_A02_02                              :=      24522       ,
	PRECISOR_UR_A03_01                              :=      24531       ,
	PRECISOR_UR_A03_02                              :=      24532       ,
	PRECISOR_UR_A04_01                              :=      24541       ,
	PRECISOR_UR_A04_02                              :=      24542       ,
	PRECISOR_UR_B01_01                              :=      24561       ,
	PRECISOR_UR_B01_02                              :=      24562       ,
	PRECISOR_UR_B02_01                              :=      24571       ,
	PRECISOR_UR_B02_02                              :=      24572       ,
	PRECISOR_UR_B03_01                              :=      24581       ,
	PRECISOR_UR_B03_02                              :=      24582       ,
	PRECISOR_UR_B04_01                              :=      24591       ,
	PRECISOR_UR_B04_02                              :=      24592       ,
	PRECISOR_UR_C01_01                              :=      24611       ,
	PRECISOR_UR_C01_02                              :=      24612       ,
	PRECISOR_UR_C02_01                              :=      24621       ,
	PRECISOR_UR_C02_02                              :=      24622       ,
	PRECISOR_UR_C03_01                              :=      24631       ,
	PRECISOR_UR_C03_02                              :=      24632       ,
	PRECISOR_UR_C04_01                              :=      24641       ,
	PRECISOR_UR_C04_02                              :=      24642       ,
	PRECISOR_UR_D01_01                              :=      24661       ,
	PRECISOR_UR_D01_02                              :=      24662       ,
	PRECISOR_UR_D02_01                              :=      24671       ,
	PRECISOR_UR_D02_02                              :=      24672       ,
	PRECISOR_UR_D03_01                              :=      24681       ,
	PRECISOR_UR_D03_02                              :=      24682       ,
	PRECISOR_UR_D04_01                              :=      24691       ,
	PRECISOR_UR_D04_02                              :=      24692       ,
	PRECISOR_DL                                     :=      25000       ,
	PRECISOR_DL_CLEAN                               :=      25001       ,
	PRECISOR_DL_01                                  :=      25002       ,
	PRECISOR_DL_02                                  :=      25003       ,
	PRECISOR_DL_CLEAN_READID                        :=      25004       ,
	PRECISOR_DL_01_READID                           :=      25005       ,
	PRECISOR_DL_02_READID                           :=      25006       ,
	PRECISOR_DL_A01_01                              :=      25011       ,
	PRECISOR_DL_A01_02                              :=      25012       ,
	PRECISOR_DL_A02_01                              :=      25021       ,
	PRECISOR_DL_A02_02                              :=      25022       ,
	PRECISOR_DL_A03_01                              :=      25031       ,
	PRECISOR_DL_A03_02                              :=      25032       ,
	PRECISOR_DL_A04_01                              :=      25041       ,
	PRECISOR_DL_A04_02                              :=      25042       ,
	PRECISOR_DL_B01_01                              :=      25061       ,
	PRECISOR_DL_B01_02                              :=      25062       ,
	PRECISOR_DL_B02_01                              :=      25071       ,
	PRECISOR_DL_B02_02                              :=      25072       ,
	PRECISOR_DL_B03_01                              :=      25081       ,
	PRECISOR_DL_B03_02                              :=      25082       ,
	PRECISOR_DL_B04_01                              :=      25091       ,
	PRECISOR_DL_B04_02                              :=      25092       ,
	PRECISOR_DL_C01_01                              :=      25111       ,
	PRECISOR_DL_C01_02                              :=      25112       ,
	PRECISOR_DL_C02_01                              :=      25121       ,
	PRECISOR_DL_C02_02                              :=      25122       ,
	PRECISOR_DL_C03_01                              :=      25131       ,
	PRECISOR_DL_C03_02                              :=      25132       ,
	PRECISOR_DL_C04_01                              :=      25141       ,
	PRECISOR_DL_C04_02                              :=      25142       ,
	PRECISOR_DL_D01_01                              :=      25161       ,
	PRECISOR_DL_D01_02                              :=      25162       ,
	PRECISOR_DL_D02_01                              :=      25171       ,
	PRECISOR_DL_D02_02                              :=      25172       ,
	PRECISOR_DL_D03_01                              :=      25181       ,
	PRECISOR_DL_D03_02                              :=      25182       ,
	PRECISOR_DL_D04_01                              :=      25191       ,
	PRECISOR_DL_D04_02                              :=      25192       ,
	PRECISOR_DR                                     :=      25500       ,
	PRECISOR_DR_CLEAN                               :=      25501       ,
	PRECISOR_DR_01                                  :=      25502       ,
	PRECISOR_DR_02                                  :=      25503       ,
	PRECISOR_DR_CLEAN_READID                        :=      25504       ,
	PRECISOR_DR_01_READID                           :=      25505       ,
	PRECISOR_DR_02_READID                           :=      25506       ,
	PRECISOR_DR_A01_01                              :=      25511       ,
	PRECISOR_DR_A01_02                              :=      25512       ,
	PRECISOR_DR_A02_01                              :=      25521       ,
	PRECISOR_DR_A02_02                              :=      25522       ,
	PRECISOR_DR_A03_01                              :=      25531       ,
	PRECISOR_DR_A03_02                              :=      25532       ,
	PRECISOR_DR_A04_01                              :=      25541       ,
	PRECISOR_DR_A04_02                              :=      25542       ,
	PRECISOR_DR_B01_01                              :=      25561       ,
	PRECISOR_DR_B01_02                              :=      25562       ,
	PRECISOR_DR_B02_01                              :=      25571       ,
	PRECISOR_DR_B02_02                              :=      25572       ,
	PRECISOR_DR_B03_01                              :=      25581       ,
	PRECISOR_DR_B03_02                              :=      25582       ,
	PRECISOR_DR_B04_01                              :=      25591       ,
	PRECISOR_DR_B04_02                              :=      25592       ,
	PRECISOR_DR_C01_01                              :=      25611       ,
	PRECISOR_DR_C01_02                              :=      25612       ,
	PRECISOR_DR_C02_01                              :=      25621       ,
	PRECISOR_DR_C02_02                              :=      25622       ,
	PRECISOR_DR_C03_01                              :=      25631       ,
	PRECISOR_DR_C03_02                              :=      25632       ,
	PRECISOR_DR_C04_01                              :=      25641       ,
	PRECISOR_DR_C04_02                              :=      25642       ,
	PRECISOR_DR_D01_01                              :=      25661       ,
	PRECISOR_DR_D01_02                              :=      25662       ,
	PRECISOR_DR_D02_01                              :=      25671       ,
	PRECISOR_DR_D02_02                              :=      25672       ,
	PRECISOR_DR_D03_01                              :=      25681       ,
	PRECISOR_DR_D03_02                              :=      25682       ,
	PRECISOR_DR_D04_01                              :=      25691       ,
	PRECISOR_DR_D04_02                              :=      25692       ,
	TBOT_L                                          :=      30000       ,
	TBOT_L_RFID                                     :=      30001       ,
	TBOT_L_SERVICE                                  :=      30002       ,
	TBOT_L_PARK                                     :=      30003       ,
	TBOT_L_HEAD_A01                                 :=      30020       ,
	TBOT_L_HEAD_A02                                 :=      30040       ,
	TBOT_L_HEAD_A03                                 :=      30060       ,
	TBOT_L_HEAD_A04                                 :=      30080       ,
	TBOT_L_HEAD_B01                                 :=      30100       ,
	TBOT_L_HEAD_B02                                 :=      30120       ,
	TBOT_L_HEAD_B03                                 :=      30140       ,
	TBOT_L_HEAD_B04                                 :=      30160       ,
	TBOT_L_HEAD_C01                                 :=      30180       ,
	TBOT_L_HEAD_C02                                 :=      30200       ,
	TBOT_L_HEAD_C03                                 :=      30220       ,
	TBOT_L_HEAD_C04                                 :=      30240       ,
	TBOT_L_HEAD_D01                                 :=      30260       ,
	TBOT_L_HEAD_D02                                 :=      30280       ,
	TBOT_L_HEAD_D03                                 :=      30300       ,
	TBOT_L_HEAD_D04                                 :=      30320       ,
	TBOT_R                                          :=      30500       ,
	TBOT_R_RFID                                     :=      30501       ,
	TBOT_R_SERVICE                                  :=      30502       ,
	TBOT_R_PARK                                     :=      30503       ,
	TBOT_R_HEAD_A01                                 :=      30520       ,
	TBOT_R_HEAD_A02                                 :=      30540       ,
	TBOT_R_HEAD_A03                                 :=      30560       ,
	TBOT_R_HEAD_A04                                 :=      30580       ,
	TBOT_R_HEAD_B01                                 :=      30600       ,
	TBOT_R_HEAD_B02                                 :=      30620       ,
	TBOT_R_HEAD_B03                                 :=      30640       ,
	TBOT_R_HEAD_B04                                 :=      30660       ,
	TBOT_R_HEAD_C01                                 :=      30680       ,
	TBOT_R_HEAD_C02                                 :=      30700       ,
	TBOT_R_HEAD_C03                                 :=      30720       ,
	TBOT_R_HEAD_C04                                 :=      30740       ,
	TBOT_R_HEAD_D01                                 :=      30760       ,
	TBOT_R_HEAD_D02                                 :=      30780       ,
	TBOT_R_HEAD_D03                                 :=      30800       ,
	TBOT_R_HEAD_D04                                 :=      30820       ,
	COLUMN_LA                                       :=      35000       ,
	COLUMN_LB                                       :=      35100       ,
	COLUMN_LC                                       :=      35200       ,
	COLUMN_RA                                       :=      35300       ,
	COLUMN_RB                                       :=      35400       ,
	COLUMN_RC                                       :=      35500       ,
	LEVEL_LA01                                      :=      36000       ,
	LEVEL_LA02                                      :=      36010       ,
	LEVEL_LA03                                      :=      36020       ,
	LEVEL_LA04                                      :=      36030       ,
	LEVEL_LA05                                      :=      36040       ,
	LEVEL_LA06                                      :=      36050       ,
	LEVEL_LB01                                      :=      36060       ,
	LEVEL_LB02                                      :=      36070       ,
	LEVEL_LB03                                      :=      36080       ,
	LEVEL_LB04                                      :=      36090       ,
	LEVEL_LB05                                      :=      36100       ,
	LEVEL_LB06                                      :=      36110       ,
	LEVEL_LC01                                      :=      36120       ,
	LEVEL_LC02                                      :=      36130       ,
	LEVEL_LC03                                      :=      36140       ,
	LEVEL_LC04                                      :=      36150       ,
	LEVEL_LC05                                      :=      36160       ,
	LEVEL_LC06                                      :=      36170       ,
	LEVEL_RA01                                      :=      37000       ,
	LEVEL_RA02                                      :=      37010       ,
	LEVEL_RA03                                      :=      37020       ,
	LEVEL_RA04                                      :=      37030       ,
	LEVEL_RA05                                      :=      37040       ,
	LEVEL_RA06                                      :=      37050       ,
	LEVEL_RB01                                      :=      37060       ,
	LEVEL_RB02                                      :=      37070       ,
	LEVEL_RB03                                      :=      37080       ,
	LEVEL_RB04                                      :=      37090       ,
	LEVEL_RB05                                      :=      37100       ,
	LEVEL_RB06                                      :=      37110       ,
	LEVEL_RC01                                      :=      37120       ,
	LEVEL_RC02                                      :=      37130       ,
	LEVEL_RC03                                      :=      37140       ,
	LEVEL_RC04                                      :=      37150       ,
	LEVEL_RC05                                      :=      37160       ,
	LEVEL_RC06                                      :=      37170       ,
	CELL_LA101_TESTER                               :=      45000       ,
	CELL_LA101_TESTER_SOCKET_A01                    :=      45001       ,
	CELL_LA101_TESTER_SOCKET_A02                    :=      45002       ,
	CELL_LA101_TESTER_SOCKET_A03                    :=      45003       ,
	CELL_LA101_TESTER_SOCKET_A04                    :=      45004       ,
	CELL_LA101_TESTER_SOCKET_B01                    :=      45011       ,
	CELL_LA101_TESTER_SOCKET_B02                    :=      45012       ,
	CELL_LA101_TESTER_SOCKET_B03                    :=      45013       ,
	CELL_LA101_TESTER_SOCKET_B04                    :=      45014       ,
	CELL_LA101_TESTER_SOCKET_C01                    :=      45021       ,
	CELL_LA101_TESTER_SOCKET_C02                    :=      45022       ,
	CELL_LA101_TESTER_SOCKET_C03                    :=      45023       ,
	CELL_LA101_TESTER_SOCKET_C04                    :=      45024       ,
	CELL_LA101_TESTER_SOCKET_D01                    :=      45031       ,
	CELL_LA101_TESTER_SOCKET_D02                    :=      45032       ,
	CELL_LA101_TESTER_SOCKET_D03                    :=      45033       ,
	CELL_LA101_TESTER_SOCKET_D04                    :=      45034       ,
	CELL_LA101_AP                                   :=      45050       ,
	CELL_LA101_AP_TH_A01                            :=      45051       ,
	CELL_LA101_AP_TH_A02                            :=      45052       ,
	CELL_LA101_AP_TH_A03                            :=      45053       ,
	CELL_LA101_AP_TH_A04                            :=      45054       ,
	CELL_LA101_AP_TH_B01                            :=      45061       ,
	CELL_LA101_AP_TH_B02                            :=      45062       ,
	CELL_LA101_AP_TH_B03                            :=      45063       ,
	CELL_LA101_AP_TH_B04                            :=      45064       ,
	CELL_LA101_AP_TH_C01                            :=      45071       ,
	CELL_LA101_AP_TH_C02                            :=      45072       ,
	CELL_LA101_AP_TH_C03                            :=      45073       ,
	CELL_LA101_AP_TH_C04                            :=      45074       ,
	CELL_LA101_AP_TH_D01                            :=      45081       ,
	CELL_LA101_AP_TH_D02                            :=      45082       ,
	CELL_LA101_AP_TH_D03                            :=      45083       ,
	CELL_LA101_AP_TH_D04                            :=      45084       ,
	CELL_LA201_TESTER                               :=      45100       ,
	CELL_LA201_TESTER_SOCKET_A01                    :=      45101       ,
	CELL_LA201_TESTER_SOCKET_A02                    :=      45102       ,
	CELL_LA201_TESTER_SOCKET_A03                    :=      45103       ,
	CELL_LA201_TESTER_SOCKET_A04                    :=      45104       ,
	CELL_LA201_TESTER_SOCKET_B01                    :=      45111       ,
	CELL_LA201_TESTER_SOCKET_B02                    :=      45112       ,
	CELL_LA201_TESTER_SOCKET_B03                    :=      45113       ,
	CELL_LA201_TESTER_SOCKET_B04                    :=      45114       ,
	CELL_LA201_TESTER_SOCKET_C01                    :=      45121       ,
	CELL_LA201_TESTER_SOCKET_C02                    :=      45122       ,
	CELL_LA201_TESTER_SOCKET_C03                    :=      45123       ,
	CELL_LA201_TESTER_SOCKET_C04                    :=      45124       ,
	CELL_LA201_TESTER_SOCKET_D01                    :=      45131       ,
	CELL_LA201_TESTER_SOCKET_D02                    :=      45132       ,
	CELL_LA201_TESTER_SOCKET_D03                    :=      45133       ,
	CELL_LA201_TESTER_SOCKET_D04                    :=      45134       ,
	CELL_LA201_AP                                   :=      45150       ,
	CELL_LA201_AP_TH_A01                            :=      45151       ,
	CELL_LA201_AP_TH_A02                            :=      45152       ,
	CELL_LA201_AP_TH_A03                            :=      45153       ,
	CELL_LA201_AP_TH_A04                            :=      45154       ,
	CELL_LA201_AP_TH_B01                            :=      45161       ,
	CELL_LA201_AP_TH_B02                            :=      45162       ,
	CELL_LA201_AP_TH_B03                            :=      45163       ,
	CELL_LA201_AP_TH_B04                            :=      45164       ,
	CELL_LA201_AP_TH_C01                            :=      45171       ,
	CELL_LA201_AP_TH_C02                            :=      45172       ,
	CELL_LA201_AP_TH_C03                            :=      45173       ,
	CELL_LA201_AP_TH_C04                            :=      45174       ,
	CELL_LA201_AP_TH_D01                            :=      45181       ,
	CELL_LA201_AP_TH_D02                            :=      45182       ,
	CELL_LA201_AP_TH_D03                            :=      45183       ,
	CELL_LA201_AP_TH_D04                            :=      45184       ,
	CELL_LA301_TESTER                               :=      45200       ,
	CELL_LA301_TESTER_SOCKET_A01                    :=      45201       ,
	CELL_LA301_TESTER_SOCKET_A02                    :=      45202       ,
	CELL_LA301_TESTER_SOCKET_A03                    :=      45203       ,
	CELL_LA301_TESTER_SOCKET_A04                    :=      45204       ,
	CELL_LA301_TESTER_SOCKET_B01                    :=      45211       ,
	CELL_LA301_TESTER_SOCKET_B02                    :=      45212       ,
	CELL_LA301_TESTER_SOCKET_B03                    :=      45213       ,
	CELL_LA301_TESTER_SOCKET_B04                    :=      45214       ,
	CELL_LA301_TESTER_SOCKET_C01                    :=      45221       ,
	CELL_LA301_TESTER_SOCKET_C02                    :=      45222       ,
	CELL_LA301_TESTER_SOCKET_C03                    :=      45223       ,
	CELL_LA301_TESTER_SOCKET_C04                    :=      45224       ,
	CELL_LA301_TESTER_SOCKET_D01                    :=      45231       ,
	CELL_LA301_TESTER_SOCKET_D02                    :=      45232       ,
	CELL_LA301_TESTER_SOCKET_D03                    :=      45233       ,
	CELL_LA301_TESTER_SOCKET_D04                    :=      45234       ,
	CELL_LA301_AP                                   :=      45250       ,
	CELL_LA301_AP_TH_A01                            :=      45251       ,
	CELL_LA301_AP_TH_A02                            :=      45252       ,
	CELL_LA301_AP_TH_A03                            :=      45253       ,
	CELL_LA301_AP_TH_A04                            :=      45254       ,
	CELL_LA301_AP_TH_B01                            :=      45261       ,
	CELL_LA301_AP_TH_B02                            :=      45262       ,
	CELL_LA301_AP_TH_B03                            :=      45263       ,
	CELL_LA301_AP_TH_B04                            :=      45264       ,
	CELL_LA301_AP_TH_C01                            :=      45271       ,
	CELL_LA301_AP_TH_C02                            :=      45272       ,
	CELL_LA301_AP_TH_C03                            :=      45273       ,
	CELL_LA301_AP_TH_C04                            :=      45274       ,
	CELL_LA301_AP_TH_D01                            :=      45281       ,
	CELL_LA301_AP_TH_D02                            :=      45282       ,
	CELL_LA301_AP_TH_D03                            :=      45283       ,
	CELL_LA301_AP_TH_D04                            :=      45284       ,
	CELL_LA401_TESTER                               :=      45300       ,
	CELL_LA401_TESTER_SOCKET_A01                    :=      45301       ,
	CELL_LA401_TESTER_SOCKET_A02                    :=      45302       ,
	CELL_LA401_TESTER_SOCKET_A03                    :=      45303       ,
	CELL_LA401_TESTER_SOCKET_A04                    :=      45304       ,
	CELL_LA401_TESTER_SOCKET_B01                    :=      45311       ,
	CELL_LA401_TESTER_SOCKET_B02                    :=      45312       ,
	CELL_LA401_TESTER_SOCKET_B03                    :=      45313       ,
	CELL_LA401_TESTER_SOCKET_B04                    :=      45314       ,
	CELL_LA401_TESTER_SOCKET_C01                    :=      45321       ,
	CELL_LA401_TESTER_SOCKET_C02                    :=      45322       ,
	CELL_LA401_TESTER_SOCKET_C03                    :=      45323       ,
	CELL_LA401_TESTER_SOCKET_C04                    :=      45324       ,
	CELL_LA401_TESTER_SOCKET_D01                    :=      45331       ,
	CELL_LA401_TESTER_SOCKET_D02                    :=      45332       ,
	CELL_LA401_TESTER_SOCKET_D03                    :=      45333       ,
	CELL_LA401_TESTER_SOCKET_D04                    :=      45334       ,
	CELL_LA401_AP                                   :=      45350       ,
	CELL_LA401_AP_TH_A01                            :=      45351       ,
	CELL_LA401_AP_TH_A02                            :=      45352       ,
	CELL_LA401_AP_TH_A03                            :=      45353       ,
	CELL_LA401_AP_TH_A04                            :=      45354       ,
	CELL_LA401_AP_TH_B01                            :=      45361       ,
	CELL_LA401_AP_TH_B02                            :=      45362       ,
	CELL_LA401_AP_TH_B03                            :=      45363       ,
	CELL_LA401_AP_TH_B04                            :=      45364       ,
	CELL_LA401_AP_TH_C01                            :=      45371       ,
	CELL_LA401_AP_TH_C02                            :=      45372       ,
	CELL_LA401_AP_TH_C03                            :=      45373       ,
	CELL_LA401_AP_TH_C04                            :=      45374       ,
	CELL_LA401_AP_TH_D01                            :=      45381       ,
	CELL_LA401_AP_TH_D02                            :=      45382       ,
	CELL_LA401_AP_TH_D03                            :=      45383       ,
	CELL_LA401_AP_TH_D04                            :=      45384       ,
	CELL_LA501_TESTER                               :=      45400       ,
	CELL_LA501_TESTER_SOCKET_A01                    :=      45401       ,
	CELL_LA501_TESTER_SOCKET_A02                    :=      45402       ,
	CELL_LA501_TESTER_SOCKET_A03                    :=      45403       ,
	CELL_LA501_TESTER_SOCKET_A04                    :=      45404       ,
	CELL_LA501_TESTER_SOCKET_B01                    :=      45411       ,
	CELL_LA501_TESTER_SOCKET_B02                    :=      45412       ,
	CELL_LA501_TESTER_SOCKET_B03                    :=      45413       ,
	CELL_LA501_TESTER_SOCKET_B04                    :=      45414       ,
	CELL_LA501_TESTER_SOCKET_C01                    :=      45421       ,
	CELL_LA501_TESTER_SOCKET_C02                    :=      45422       ,
	CELL_LA501_TESTER_SOCKET_C03                    :=      45423       ,
	CELL_LA501_TESTER_SOCKET_C04                    :=      45424       ,
	CELL_LA501_TESTER_SOCKET_D01                    :=      45431       ,
	CELL_LA501_TESTER_SOCKET_D02                    :=      45432       ,
	CELL_LA501_TESTER_SOCKET_D03                    :=      45433       ,
	CELL_LA501_TESTER_SOCKET_D04                    :=      45434       ,
	CELL_LA501_AP                                   :=      45450       ,
	CELL_LA501_AP_TH_A01                            :=      45451       ,
	CELL_LA501_AP_TH_A02                            :=      45452       ,
	CELL_LA501_AP_TH_A03                            :=      45453       ,
	CELL_LA501_AP_TH_A04                            :=      45454       ,
	CELL_LA501_AP_TH_B01                            :=      45461       ,
	CELL_LA501_AP_TH_B02                            :=      45462       ,
	CELL_LA501_AP_TH_B03                            :=      45463       ,
	CELL_LA501_AP_TH_B04                            :=      45464       ,
	CELL_LA501_AP_TH_C01                            :=      45471       ,
	CELL_LA501_AP_TH_C02                            :=      45472       ,
	CELL_LA501_AP_TH_C03                            :=      45473       ,
	CELL_LA501_AP_TH_C04                            :=      45474       ,
	CELL_LA501_AP_TH_D01                            :=      45481       ,
	CELL_LA501_AP_TH_D02                            :=      45482       ,
	CELL_LA501_AP_TH_D03                            :=      45483       ,
	CELL_LA501_AP_TH_D04                            :=      45484       ,
	CELL_LA601_TESTER                               :=      45500       ,
	CELL_LA601_TESTER_SOCKET_A01                    :=      45501       ,
	CELL_LA601_TESTER_SOCKET_A02                    :=      45502       ,
	CELL_LA601_TESTER_SOCKET_A03                    :=      45503       ,
	CELL_LA601_TESTER_SOCKET_A04                    :=      45504       ,
	CELL_LA601_TESTER_SOCKET_B01                    :=      45511       ,
	CELL_LA601_TESTER_SOCKET_B02                    :=      45512       ,
	CELL_LA601_TESTER_SOCKET_B03                    :=      45513       ,
	CELL_LA601_TESTER_SOCKET_B04                    :=      45514       ,
	CELL_LA601_TESTER_SOCKET_C01                    :=      45521       ,
	CELL_LA601_TESTER_SOCKET_C02                    :=      45522       ,
	CELL_LA601_TESTER_SOCKET_C03                    :=      45523       ,
	CELL_LA601_TESTER_SOCKET_C04                    :=      45524       ,
	CELL_LA601_TESTER_SOCKET_D01                    :=      45531       ,
	CELL_LA601_TESTER_SOCKET_D02                    :=      45532       ,
	CELL_LA601_TESTER_SOCKET_D03                    :=      45533       ,
	CELL_LA601_TESTER_SOCKET_D04                    :=      45534       ,
	CELL_LA601_AP                                   :=      45550       ,
	CELL_LA601_AP_TH_A01                            :=      45551       ,
	CELL_LA601_AP_TH_A02                            :=      45552       ,
	CELL_LA601_AP_TH_A03                            :=      45553       ,
	CELL_LA601_AP_TH_A04                            :=      45554       ,
	CELL_LA601_AP_TH_B01                            :=      45561       ,
	CELL_LA601_AP_TH_B02                            :=      45562       ,
	CELL_LA601_AP_TH_B03                            :=      45563       ,
	CELL_LA601_AP_TH_B04                            :=      45564       ,
	CELL_LA601_AP_TH_C01                            :=      45571       ,
	CELL_LA601_AP_TH_C02                            :=      45572       ,
	CELL_LA601_AP_TH_C03                            :=      45573       ,
	CELL_LA601_AP_TH_C04                            :=      45574       ,
	CELL_LA601_AP_TH_D01                            :=      45581       ,
	CELL_LA601_AP_TH_D02                            :=      45582       ,
	CELL_LA601_AP_TH_D03                            :=      45583       ,
	CELL_LA601_AP_TH_D04                            :=      45584       ,
	CELL_LB101_TESTER                               :=      46000       ,
	CELL_LB101_TESTER_SOCKET_A01                    :=      46001       ,
	CELL_LB101_TESTER_SOCKET_A02                    :=      46002       ,
	CELL_LB101_TESTER_SOCKET_A03                    :=      46003       ,
	CELL_LB101_TESTER_SOCKET_A04                    :=      46004       ,
	CELL_LB101_TESTER_SOCKET_B01                    :=      46011       ,
	CELL_LB101_TESTER_SOCKET_B02                    :=      46012       ,
	CELL_LB101_TESTER_SOCKET_B03                    :=      46013       ,
	CELL_LB101_TESTER_SOCKET_B04                    :=      46014       ,
	CELL_LB101_TESTER_SOCKET_C01                    :=      46021       ,
	CELL_LB101_TESTER_SOCKET_C02                    :=      46022       ,
	CELL_LB101_TESTER_SOCKET_C03                    :=      46023       ,
	CELL_LB101_TESTER_SOCKET_C04                    :=      46024       ,
	CELL_LB101_TESTER_SOCKET_D01                    :=      46031       ,
	CELL_LB101_TESTER_SOCKET_D02                    :=      46032       ,
	CELL_LB101_TESTER_SOCKET_D03                    :=      46033       ,
	CELL_LB101_TESTER_SOCKET_D04                    :=      46034       ,
	CELL_LB101_AP                                   :=      46050       ,
	CELL_LB101_AP_TH_A01                            :=      46051       ,
	CELL_LB101_AP_TH_A02                            :=      46052       ,
	CELL_LB101_AP_TH_A03                            :=      46053       ,
	CELL_LB101_AP_TH_A04                            :=      46054       ,
	CELL_LB101_AP_TH_B01                            :=      46061       ,
	CELL_LB101_AP_TH_B02                            :=      46062       ,
	CELL_LB101_AP_TH_B03                            :=      46063       ,
	CELL_LB101_AP_TH_B04                            :=      46064       ,
	CELL_LB101_AP_TH_C01                            :=      46071       ,
	CELL_LB101_AP_TH_C02                            :=      46072       ,
	CELL_LB101_AP_TH_C03                            :=      46073       ,
	CELL_LB101_AP_TH_C04                            :=      46074       ,
	CELL_LB101_AP_TH_D01                            :=      46081       ,
	CELL_LB101_AP_TH_D02                            :=      46082       ,
	CELL_LB101_AP_TH_D03                            :=      46083       ,
	CELL_LB101_AP_TH_D04                            :=      46084       ,
	CELL_LB201_TESTER                               :=      46100       ,
	CELL_LB201_TESTER_SOCKET_A01                    :=      46101       ,
	CELL_LB201_TESTER_SOCKET_A02                    :=      46102       ,
	CELL_LB201_TESTER_SOCKET_A03                    :=      46103       ,
	CELL_LB201_TESTER_SOCKET_A04                    :=      46104       ,
	CELL_LB201_TESTER_SOCKET_B01                    :=      46111       ,
	CELL_LB201_TESTER_SOCKET_B02                    :=      46112       ,
	CELL_LB201_TESTER_SOCKET_B03                    :=      46113       ,
	CELL_LB201_TESTER_SOCKET_B04                    :=      46114       ,
	CELL_LB201_TESTER_SOCKET_C01                    :=      46121       ,
	CELL_LB201_TESTER_SOCKET_C02                    :=      46122       ,
	CELL_LB201_TESTER_SOCKET_C03                    :=      46123       ,
	CELL_LB201_TESTER_SOCKET_C04                    :=      46124       ,
	CELL_LB201_TESTER_SOCKET_D01                    :=      46131       ,
	CELL_LB201_TESTER_SOCKET_D02                    :=      46132       ,
	CELL_LB201_TESTER_SOCKET_D03                    :=      46133       ,
	CELL_LB201_TESTER_SOCKET_D04                    :=      46134       ,
	CELL_LB201_AP                                   :=      46150       ,
	CELL_LB201_AP_TH_A01                            :=      46151       ,
	CELL_LB201_AP_TH_A02                            :=      46152       ,
	CELL_LB201_AP_TH_A03                            :=      46153       ,
	CELL_LB201_AP_TH_A04                            :=      46154       ,
	CELL_LB201_AP_TH_B01                            :=      46161       ,
	CELL_LB201_AP_TH_B02                            :=      46162       ,
	CELL_LB201_AP_TH_B03                            :=      46163       ,
	CELL_LB201_AP_TH_B04                            :=      46164       ,
	CELL_LB201_AP_TH_C01                            :=      46171       ,
	CELL_LB201_AP_TH_C02                            :=      46172       ,
	CELL_LB201_AP_TH_C03                            :=      46173       ,
	CELL_LB201_AP_TH_C04                            :=      46174       ,
	CELL_LB201_AP_TH_D01                            :=      46181       ,
	CELL_LB201_AP_TH_D02                            :=      46182       ,
	CELL_LB201_AP_TH_D03                            :=      46183       ,
	CELL_LB201_AP_TH_D04                            :=      46184       ,
	CELL_LB301_TESTER                               :=      46200       ,
	CELL_LB301_TESTER_SOCKET_A01                    :=      46201       ,
	CELL_LB301_TESTER_SOCKET_A02                    :=      46202       ,
	CELL_LB301_TESTER_SOCKET_A03                    :=      46203       ,
	CELL_LB301_TESTER_SOCKET_A04                    :=      46204       ,
	CELL_LB301_TESTER_SOCKET_B01                    :=      46211       ,
	CELL_LB301_TESTER_SOCKET_B02                    :=      46212       ,
	CELL_LB301_TESTER_SOCKET_B03                    :=      46213       ,
	CELL_LB301_TESTER_SOCKET_B04                    :=      46214       ,
	CELL_LB301_TESTER_SOCKET_C01                    :=      46221       ,
	CELL_LB301_TESTER_SOCKET_C02                    :=      46222       ,
	CELL_LB301_TESTER_SOCKET_C03                    :=      46223       ,
	CELL_LB301_TESTER_SOCKET_C04                    :=      46224       ,
	CELL_LB301_TESTER_SOCKET_D01                    :=      46231       ,
	CELL_LB301_TESTER_SOCKET_D02                    :=      46232       ,
	CELL_LB301_TESTER_SOCKET_D03                    :=      46233       ,
	CELL_LB301_TESTER_SOCKET_D04                    :=      46234       ,
	CELL_LB301_AP                                   :=      46250       ,
	CELL_LB301_AP_TH_A01                            :=      46251       ,
	CELL_LB301_AP_TH_A02                            :=      46252       ,
	CELL_LB301_AP_TH_A03                            :=      46253       ,
	CELL_LB301_AP_TH_A04                            :=      46254       ,
	CELL_LB301_AP_TH_B01                            :=      46261       ,
	CELL_LB301_AP_TH_B02                            :=      46262       ,
	CELL_LB301_AP_TH_B03                            :=      46263       ,
	CELL_LB301_AP_TH_B04                            :=      46264       ,
	CELL_LB301_AP_TH_C01                            :=      46271       ,
	CELL_LB301_AP_TH_C02                            :=      46272       ,
	CELL_LB301_AP_TH_C03                            :=      46273       ,
	CELL_LB301_AP_TH_C04                            :=      46274       ,
	CELL_LB301_AP_TH_D01                            :=      46281       ,
	CELL_LB301_AP_TH_D02                            :=      46282       ,
	CELL_LB301_AP_TH_D03                            :=      46283       ,
	CELL_LB301_AP_TH_D04                            :=      46284       ,
	CELL_LB401_TESTER                               :=      46300       ,
	CELL_LB401_TESTER_SOCKET_A01                    :=      46301       ,
	CELL_LB401_TESTER_SOCKET_A02                    :=      46302       ,
	CELL_LB401_TESTER_SOCKET_A03                    :=      46303       ,
	CELL_LB401_TESTER_SOCKET_A04                    :=      46304       ,
	CELL_LB401_TESTER_SOCKET_B01                    :=      46311       ,
	CELL_LB401_TESTER_SOCKET_B02                    :=      46312       ,
	CELL_LB401_TESTER_SOCKET_B03                    :=      46313       ,
	CELL_LB401_TESTER_SOCKET_B04                    :=      46314       ,
	CELL_LB401_TESTER_SOCKET_C01                    :=      46321       ,
	CELL_LB401_TESTER_SOCKET_C02                    :=      46322       ,
	CELL_LB401_TESTER_SOCKET_C03                    :=      46323       ,
	CELL_LB401_TESTER_SOCKET_C04                    :=      46324       ,
	CELL_LB401_TESTER_SOCKET_D01                    :=      46331       ,
	CELL_LB401_TESTER_SOCKET_D02                    :=      46332       ,
	CELL_LB401_TESTER_SOCKET_D03                    :=      46333       ,
	CELL_LB401_TESTER_SOCKET_D04                    :=      46334       ,
	CELL_LB401_AP                                   :=      46350       ,
	CELL_LB401_AP_TH_A01                            :=      46351       ,
	CELL_LB401_AP_TH_A02                            :=      46352       ,
	CELL_LB401_AP_TH_A03                            :=      46353       ,
	CELL_LB401_AP_TH_A04                            :=      46354       ,
	CELL_LB401_AP_TH_B01                            :=      46361       ,
	CELL_LB401_AP_TH_B02                            :=      46362       ,
	CELL_LB401_AP_TH_B03                            :=      46363       ,
	CELL_LB401_AP_TH_B04                            :=      46364       ,
	CELL_LB401_AP_TH_C01                            :=      46371       ,
	CELL_LB401_AP_TH_C02                            :=      46372       ,
	CELL_LB401_AP_TH_C03                            :=      46373       ,
	CELL_LB401_AP_TH_C04                            :=      46374       ,
	CELL_LB401_AP_TH_D01                            :=      46381       ,
	CELL_LB401_AP_TH_D02                            :=      46382       ,
	CELL_LB401_AP_TH_D03                            :=      46383       ,
	CELL_LB401_AP_TH_D04                            :=      46384       ,
	CELL_LB501_TESTER                               :=      46400       ,
	CELL_LB501_TESTER_SOCKET_A01                    :=      46401       ,
	CELL_LB501_TESTER_SOCKET_A02                    :=      46402       ,
	CELL_LB501_TESTER_SOCKET_A03                    :=      46403       ,
	CELL_LB501_TESTER_SOCKET_A04                    :=      46404       ,
	CELL_LB501_TESTER_SOCKET_B01                    :=      46411       ,
	CELL_LB501_TESTER_SOCKET_B02                    :=      46412       ,
	CELL_LB501_TESTER_SOCKET_B03                    :=      46413       ,
	CELL_LB501_TESTER_SOCKET_B04                    :=      46414       ,
	CELL_LB501_TESTER_SOCKET_C01                    :=      46421       ,
	CELL_LB501_TESTER_SOCKET_C02                    :=      46422       ,
	CELL_LB501_TESTER_SOCKET_C03                    :=      46423       ,
	CELL_LB501_TESTER_SOCKET_C04                    :=      46424       ,
	CELL_LB501_TESTER_SOCKET_D01                    :=      46431       ,
	CELL_LB501_TESTER_SOCKET_D02                    :=      46432       ,
	CELL_LB501_TESTER_SOCKET_D03                    :=      46433       ,
	CELL_LB501_TESTER_SOCKET_D04                    :=      46434       ,
	CELL_LB501_AP                                   :=      46450       ,
	CELL_LB501_AP_TH_A01                            :=      46451       ,
	CELL_LB501_AP_TH_A02                            :=      46452       ,
	CELL_LB501_AP_TH_A03                            :=      46453       ,
	CELL_LB501_AP_TH_A04                            :=      46454       ,
	CELL_LB501_AP_TH_B01                            :=      46461       ,
	CELL_LB501_AP_TH_B02                            :=      46462       ,
	CELL_LB501_AP_TH_B03                            :=      46463       ,
	CELL_LB501_AP_TH_B04                            :=      46464       ,
	CELL_LB501_AP_TH_C01                            :=      46471       ,
	CELL_LB501_AP_TH_C02                            :=      46472       ,
	CELL_LB501_AP_TH_C03                            :=      46473       ,
	CELL_LB501_AP_TH_C04                            :=      46474       ,
	CELL_LB501_AP_TH_D01                            :=      46481       ,
	CELL_LB501_AP_TH_D02                            :=      46482       ,
	CELL_LB501_AP_TH_D03                            :=      46483       ,
	CELL_LB501_AP_TH_D04                            :=      46484       ,
	CELL_LB601_TESTER                               :=      46500       ,
	CELL_LB601_TESTER_SOCKET_A01                    :=      46501       ,
	CELL_LB601_TESTER_SOCKET_A02                    :=      46502       ,
	CELL_LB601_TESTER_SOCKET_A03                    :=      46503       ,
	CELL_LB601_TESTER_SOCKET_A04                    :=      46504       ,
	CELL_LB601_TESTER_SOCKET_B01                    :=      46511       ,
	CELL_LB601_TESTER_SOCKET_B02                    :=      46512       ,
	CELL_LB601_TESTER_SOCKET_B03                    :=      46513       ,
	CELL_LB601_TESTER_SOCKET_B04                    :=      46514       ,
	CELL_LB601_TESTER_SOCKET_C01                    :=      46521       ,
	CELL_LB601_TESTER_SOCKET_C02                    :=      46522       ,
	CELL_LB601_TESTER_SOCKET_C03                    :=      46523       ,
	CELL_LB601_TESTER_SOCKET_C04                    :=      46524       ,
	CELL_LB601_TESTER_SOCKET_D01                    :=      46531       ,
	CELL_LB601_TESTER_SOCKET_D02                    :=      46532       ,
	CELL_LB601_TESTER_SOCKET_D03                    :=      46533       ,
	CELL_LB601_TESTER_SOCKET_D04                    :=      46534       ,
	CELL_LB601_AP                                   :=      46550       ,
	CELL_LB601_AP_TH_A01                            :=      46551       ,
	CELL_LB601_AP_TH_A02                            :=      46552       ,
	CELL_LB601_AP_TH_A03                            :=      46553       ,
	CELL_LB601_AP_TH_A04                            :=      46554       ,
	CELL_LB601_AP_TH_B01                            :=      46561       ,
	CELL_LB601_AP_TH_B02                            :=      46562       ,
	CELL_LB601_AP_TH_B03                            :=      46563       ,
	CELL_LB601_AP_TH_B04                            :=      46564       ,
	CELL_LB601_AP_TH_C01                            :=      46571       ,
	CELL_LB601_AP_TH_C02                            :=      46572       ,
	CELL_LB601_AP_TH_C03                            :=      46573       ,
	CELL_LB601_AP_TH_C04                            :=      46574       ,
	CELL_LB601_AP_TH_D01                            :=      46581       ,
	CELL_LB601_AP_TH_D02                            :=      46582       ,
	CELL_LB601_AP_TH_D03                            :=      46583       ,
	CELL_LB601_AP_TH_D04                            :=      46584       ,
	CELL_LC101_TESTER                               :=      47000       ,
	CELL_LC101_TESTER_SOCKET_A01                    :=      47001       ,
	CELL_LC101_TESTER_SOCKET_A02                    :=      47002       ,
	CELL_LC101_TESTER_SOCKET_A03                    :=      47003       ,
	CELL_LC101_TESTER_SOCKET_A04                    :=      47004       ,
	CELL_LC101_TESTER_SOCKET_B01                    :=      47011       ,
	CELL_LC101_TESTER_SOCKET_B02                    :=      47012       ,
	CELL_LC101_TESTER_SOCKET_B03                    :=      47013       ,
	CELL_LC101_TESTER_SOCKET_B04                    :=      47014       ,
	CELL_LC101_TESTER_SOCKET_C01                    :=      47021       ,
	CELL_LC101_TESTER_SOCKET_C02                    :=      47022       ,
	CELL_LC101_TESTER_SOCKET_C03                    :=      47023       ,
	CELL_LC101_TESTER_SOCKET_C04                    :=      47024       ,
	CELL_LC101_TESTER_SOCKET_D01                    :=      47031       ,
	CELL_LC101_TESTER_SOCKET_D02                    :=      47032       ,
	CELL_LC101_TESTER_SOCKET_D03                    :=      47033       ,
	CELL_LC101_TESTER_SOCKET_D04                    :=      47034       ,
	CELL_LC101_AP                                   :=      47050       ,
	CELL_LC101_AP_TH_A01                            :=      47051       ,
	CELL_LC101_AP_TH_A02                            :=      47052       ,
	CELL_LC101_AP_TH_A03                            :=      47053       ,
	CELL_LC101_AP_TH_A04                            :=      47054       ,
	CELL_LC101_AP_TH_B01                            :=      47061       ,
	CELL_LC101_AP_TH_B02                            :=      47062       ,
	CELL_LC101_AP_TH_B03                            :=      47063       ,
	CELL_LC101_AP_TH_B04                            :=      47064       ,
	CELL_LC101_AP_TH_C01                            :=      47071       ,
	CELL_LC101_AP_TH_C02                            :=      47072       ,
	CELL_LC101_AP_TH_C03                            :=      47073       ,
	CELL_LC101_AP_TH_C04                            :=      47074       ,
	CELL_LC101_AP_TH_D01                            :=      47081       ,
	CELL_LC101_AP_TH_D02                            :=      47082       ,
	CELL_LC101_AP_TH_D03                            :=      47083       ,
	CELL_LC101_AP_TH_D04                            :=      47084       ,
	CELL_LC201_TESTER                               :=      47100       ,
	CELL_LC201_TESTER_SOCKET_A01                    :=      47101       ,
	CELL_LC201_TESTER_SOCKET_A02                    :=      47102       ,
	CELL_LC201_TESTER_SOCKET_A03                    :=      47103       ,
	CELL_LC201_TESTER_SOCKET_A04                    :=      47104       ,
	CELL_LC201_TESTER_SOCKET_B01                    :=      47111       ,
	CELL_LC201_TESTER_SOCKET_B02                    :=      47112       ,
	CELL_LC201_TESTER_SOCKET_B03                    :=      47113       ,
	CELL_LC201_TESTER_SOCKET_B04                    :=      47114       ,
	CELL_LC201_TESTER_SOCKET_C01                    :=      47121       ,
	CELL_LC201_TESTER_SOCKET_C02                    :=      47122       ,
	CELL_LC201_TESTER_SOCKET_C03                    :=      47123       ,
	CELL_LC201_TESTER_SOCKET_C04                    :=      47124       ,
	CELL_LC201_TESTER_SOCKET_D01                    :=      47131       ,
	CELL_LC201_TESTER_SOCKET_D02                    :=      47132       ,
	CELL_LC201_TESTER_SOCKET_D03                    :=      47133       ,
	CELL_LC201_TESTER_SOCKET_D04                    :=      47134       ,
	CELL_LC201_AP                                   :=      47150       ,
	CELL_LC201_AP_TH_A01                            :=      47151       ,
	CELL_LC201_AP_TH_A02                            :=      47152       ,
	CELL_LC201_AP_TH_A03                            :=      47153       ,
	CELL_LC201_AP_TH_A04                            :=      47154       ,
	CELL_LC201_AP_TH_B01                            :=      47161       ,
	CELL_LC201_AP_TH_B02                            :=      47162       ,
	CELL_LC201_AP_TH_B03                            :=      47163       ,
	CELL_LC201_AP_TH_B04                            :=      47164       ,
	CELL_LC201_AP_TH_C01                            :=      47171       ,
	CELL_LC201_AP_TH_C02                            :=      47172       ,
	CELL_LC201_AP_TH_C03                            :=      47173       ,
	CELL_LC201_AP_TH_C04                            :=      47174       ,
	CELL_LC201_AP_TH_D01                            :=      47181       ,
	CELL_LC201_AP_TH_D02                            :=      47182       ,
	CELL_LC201_AP_TH_D03                            :=      47183       ,
	CELL_LC201_AP_TH_D04                            :=      47184       ,
	CELL_LC301_TESTER                               :=      47200       ,
	CELL_LC301_TESTER_SOCKET_A01                    :=      47201       ,
	CELL_LC301_TESTER_SOCKET_A02                    :=      47202       ,
	CELL_LC301_TESTER_SOCKET_A03                    :=      47203       ,
	CELL_LC301_TESTER_SOCKET_A04                    :=      47204       ,
	CELL_LC301_TESTER_SOCKET_B01                    :=      47211       ,
	CELL_LC301_TESTER_SOCKET_B02                    :=      47212       ,
	CELL_LC301_TESTER_SOCKET_B03                    :=      47213       ,
	CELL_LC301_TESTER_SOCKET_B04                    :=      47214       ,
	CELL_LC301_TESTER_SOCKET_C01                    :=      47221       ,
	CELL_LC301_TESTER_SOCKET_C02                    :=      47222       ,
	CELL_LC301_TESTER_SOCKET_C03                    :=      47223       ,
	CELL_LC301_TESTER_SOCKET_C04                    :=      47224       ,
	CELL_LC301_TESTER_SOCKET_D01                    :=      47231       ,
	CELL_LC301_TESTER_SOCKET_D02                    :=      47232       ,
	CELL_LC301_TESTER_SOCKET_D03                    :=      47233       ,
	CELL_LC301_TESTER_SOCKET_D04                    :=      47234       ,
	CELL_LC301_AP                                   :=      47250       ,
	CELL_LC301_AP_TH_A01                            :=      47251       ,
	CELL_LC301_AP_TH_A02                            :=      47252       ,
	CELL_LC301_AP_TH_A03                            :=      47253       ,
	CELL_LC301_AP_TH_A04                            :=      47254       ,
	CELL_LC301_AP_TH_B01                            :=      47261       ,
	CELL_LC301_AP_TH_B02                            :=      47262       ,
	CELL_LC301_AP_TH_B03                            :=      47263       ,
	CELL_LC301_AP_TH_B04                            :=      47264       ,
	CELL_LC301_AP_TH_C01                            :=      47271       ,
	CELL_LC301_AP_TH_C02                            :=      47272       ,
	CELL_LC301_AP_TH_C03                            :=      47273       ,
	CELL_LC301_AP_TH_C04                            :=      47274       ,
	CELL_LC301_AP_TH_D01                            :=      47281       ,
	CELL_LC301_AP_TH_D02                            :=      47282       ,
	CELL_LC301_AP_TH_D03                            :=      47283       ,
	CELL_LC301_AP_TH_D04                            :=      47284       ,
	CELL_LC401_TESTER                               :=      47300       ,
	CELL_LC401_TESTER_SOCKET_A01                    :=      47301       ,
	CELL_LC401_TESTER_SOCKET_A02                    :=      47302       ,
	CELL_LC401_TESTER_SOCKET_A03                    :=      47303       ,
	CELL_LC401_TESTER_SOCKET_A04                    :=      47304       ,
	CELL_LC401_TESTER_SOCKET_B01                    :=      47311       ,
	CELL_LC401_TESTER_SOCKET_B02                    :=      47312       ,
	CELL_LC401_TESTER_SOCKET_B03                    :=      47313       ,
	CELL_LC401_TESTER_SOCKET_B04                    :=      47314       ,
	CELL_LC401_TESTER_SOCKET_C01                    :=      47321       ,
	CELL_LC401_TESTER_SOCKET_C02                    :=      47322       ,
	CELL_LC401_TESTER_SOCKET_C03                    :=      47323       ,
	CELL_LC401_TESTER_SOCKET_C04                    :=      47324       ,
	CELL_LC401_TESTER_SOCKET_D01                    :=      47331       ,
	CELL_LC401_TESTER_SOCKET_D02                    :=      47332       ,
	CELL_LC401_TESTER_SOCKET_D03                    :=      47333       ,
	CELL_LC401_TESTER_SOCKET_D04                    :=      47334       ,
	CELL_LC401_AP                                   :=      47350       ,
	CELL_LC401_AP_TH_A01                            :=      47351       ,
	CELL_LC401_AP_TH_A02                            :=      47352       ,
	CELL_LC401_AP_TH_A03                            :=      47353       ,
	CELL_LC401_AP_TH_A04                            :=      47354       ,
	CELL_LC401_AP_TH_B01                            :=      47361       ,
	CELL_LC401_AP_TH_B02                            :=      47362       ,
	CELL_LC401_AP_TH_B03                            :=      47363       ,
	CELL_LC401_AP_TH_B04                            :=      47364       ,
	CELL_LC401_AP_TH_C01                            :=      47371       ,
	CELL_LC401_AP_TH_C02                            :=      47372       ,
	CELL_LC401_AP_TH_C03                            :=      47373       ,
	CELL_LC401_AP_TH_C04                            :=      47374       ,
	CELL_LC401_AP_TH_D01                            :=      47381       ,
